INTERFACE IDevice

METHOD turnOn
VAR_INPUT
END_VAR
END_METHOD

END_INTERFACE

(* stored: Version 1.1.0.1, ProductVersion 3.1.4024.11
   Itf IDevice: Id {3b96e9e2-9c67-472d-b9ed-509e4768d499}
   Method turnOn: Id {cc1a2356-bc53-4200-9a48-a27221f86448} *)
